// Mitsubishi GX Works2 project: 14-06-2020 LAB 2_Sequence_2   PLC: FX3G

PROGRAM MAIN
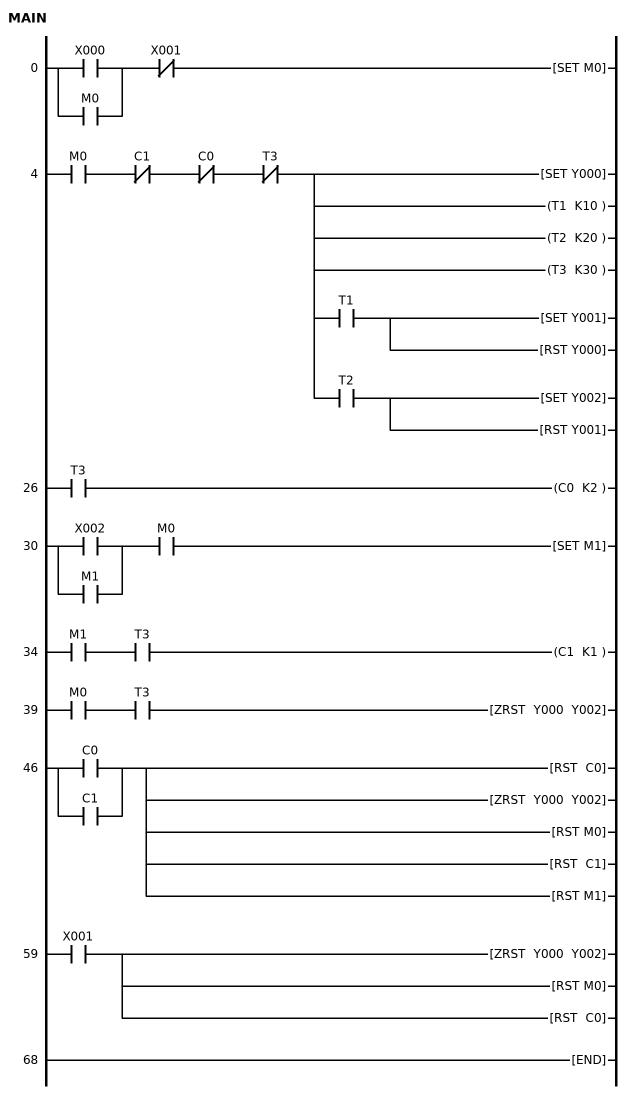
0     LD      X000
      OR      M0
      ANI     X001
      SET     M0
4     LD      M0
      ANI     C1
      ANI     C0
      ANI     T3
      SET     Y000
      OUT     T1 K10
      OUT     T2 K20
      OUT     T3 K30
      MPS
      AND     T1
      SET     Y001
      RST     Y000
      MPP
      AND     T2
      SET     Y002
      RST     Y001
26    LD      T3
      OUT     C0 K2
30    LD      X002
      OR      M1
      AND     M0
      SET     M1
34    LD      M1
      AND     T3
      OUT     C1 K1
39    LD      M0
      AND     T3
      ZRST    Y000 Y002
46    LD      C0
      OR      C1
      RST     C0
      ZRST    Y000 Y002
      RST     M0
      RST     C1
      RST     M1
59    LD      X001
      ZRST    Y000 Y002
      RST     M0
      RST     C0
68    END
END_PROGRAM
